(*
A list implementation for managing `I_Component`.  
*)
INTERFACE I_CompList EXTENDS I_Debug

(*
Provides the maximum capacity of the list.
*)
PROPERTY Cap : UDINT
GET
END_GET
END_PROPERTY

(*
Retrieves the `I_Component` at the specified index.  
Returns:
- `Ok` - Successfully retrieves the `I_Component`.
- `Err.Idx` - The specified index is out of bounds.
- `Err.InvRef` - Invalid output reference.
- `Err.Idx` - `iOut` = 0.
*)
METHOD Get : Result
VAR_INPUT
	nIndex		: UDINT;
	iOut		: REFERENCE TO I_Component;
END_VAR
END_METHOD

END_INTERFACE

(* stored: Version 1.1.0.1
   Itf I_CompList: Id {d8fd80a0-3272-49d8-a5be-503482b9faa2}
   Property Cap: Id {3a8007cf-60c7-4ef3-aae4-3192a2117f2f}
   Get Get: Id {19a163f9-a458-498d-8c9b-c786fe2947bc}
   Method Get: Id {dfc16f17-53e4-4e50-863c-21dfe530b4b4} *)
